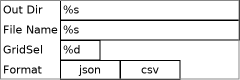
VISUALIZATION _VISU_CTGridExporter  // 240x80
VAR_IN_OUT
		mInst : FB_GridDataExporter;
END_VAR
    Rectangle (0,40 60x20), "GridSel"
    Rectangle (0,0 60x20), "Out Dir"
    Rectangle (0,60 60x20), "Format"
    RoundedRectangle (60,60 60x20), "json", colour toggle: mInst.sFileFormat = 'json'
        OnMouseClick: execute { mInst.sFileFormat := 'json'; }
    RoundedRectangle (120,60 60x20), "csv", colour toggle: mInst.sFileFormat = 'csv'
        OnMouseClick: execute { mInst.sFileFormat := 'csv'; }
    Rectangle (0,20 60x20), "File Name"
    Rectangle (60,40 40x20), "%d", text variable: mInst.nSelectGrid
        OnMouseClick: write the text variable via Default
    Rectangle (60,0 180x20), "%s", tooltip "%s", text variable: mInst.sOutputDir
        p4168582468: mInst.sOutputDir
        OnMouseClick: write the text variable via Default
    Rectangle (60,20 180x20), "%s", tooltip "%s", text variable: mInst.sFileName
        p4168582468: mInst.sFileName
        OnMouseClick: write the text variable via Default
END_VISUALIZATION

(* stored: Version 1.1.0.1, ProductVersion 3.1.4024.11
   Visu _VISU_CTGridExporter: Id {5e1a5691-10e6-41ff-8ea0-92971077d41a} *)
